FUNCTION_BLOCK Test_TExecutionWhenBusy_SetDone_SetsDone EXTENDS TUnitTestbase
VAR
    Execution : TExecution;
END_VAR

// Setup...
Execution.FB_init(
    bInitRetains := FALSE,
    bInCopyCode  := FALSE);

// Test...
Execution.Start();
Execution.SetBusy();
Execution.SetDone();

Assertion.AssertEquals_BOOL(
    Expected := TRUE,
    Actual   := Execution.Done,
    VariableName  := 'Execution.Done');

Assertion.AssertEquals_BOOL(
    Expected := TRUE,
    Actual   := Execution.Ready,
    VariableName  := 'Execution.Ready');

TestFinished();

END_FUNCTION_BLOCK

(* stored: Version 1.1.0.1, ProductVersion 3.1.4024.4
   POU Test_TExecutionWhenBusy_SetDone_SetsDone: Id {c591c302-0934-4fe7-b2fa-cb1b02a9a953}, SpecialFunc None *)
